// TIA Portal V20 export
DATA_BLOCK "CenstralShifter_Diag"   // DB43
{ S7_Optimized_Access := 'TRUE' }
// stored: MemoryReserve 100
   VAR
      Error_num_CS_PL : DInt;
      Error_num_CS_PP : DInt;
      Error_num_CS_TL : DInt;
      Error_num_CS_TP : DInt;
   END_VAR
BEGIN
END_DATA_BLOCK
